// TIA Portal V19 export
DATA_BLOCK "ControlNodes"   // DB60
// stored: MemoryReserve 100, Namespace Unit.Em1
   VAR
      em { ExternalWritable := 'False'} : "LAF_typeEmControlNode";
      jobs { ExternalWritable := 'False'} : "LAF_typeJobs";
      sequence { ExternalWritable := 'False'} : "LAF_typeSequence";
   END_VAR
BEGIN
   em.status.enabled := true;
END_DATA_BLOCK
